Universal Robots PolyScope program: LE02_50.urp

Program LE02_50 (installation=default directory=/programs/LE createdIn=5.7.0.90932 lastSavedIn=5.9.1.1031110 robotSerialNumber=20195501059)
Calibrated DH parameters: a=[0.000146, -0.418764, -0.053981, 0.000058, -0.000023, 0]; d=[0.162545, 37.319448, -206.067439, 168.881546, 0.09955, 0.099464]; alpha=[1.57004, -0.001979, 0.002304, 1.570607, -1.57066, 0]; deltaTheta=[0, -0.174616, -1.258233, 1.432844, -0.000001, 0]
BeforeStart
  'Rev 2021_12_02am 01'
  URCap Gripper Activate (Robotiq_Grippers, Robotiq Inc.) dataModel(ResetAndActivateKey=false)
  start_pose := get_actual_tcp_pose()
  MoveJ speed 60 deg/s, acceleration 80 deg/s^2 (useActiveTCP=true) feature=Base
    Waypoint Waypoint (Variable): variable=start_pose
Robot Program (runOnlyOnce=true)
  'Rev 2021_12_02am 01'
  MoveL speed 250 mm/s, acceleration 1200 mm/s^2 (useActiveTCP=true) feature=Base
    Waypoint Vertical_1: TCP in base x=296.586 y=-399.638 z=157.461 mm, rx=0.0001 ry=0 rz=-0.0068 rad; joints [110.998, -87.379, 110.673, -113.28, 270.04, 201.399] deg; TCP offset x=0 y=0 z=175 mm, rx=3.1416 ry=0 rz=0 rad
    Waypoint Tilted_2: TCP in base x=296.604 y=-399.668 z=157.504 mm, rx=-0.5593 ry=0.007 rz=-0.0068 rad; joints [119.721, -93.557, 131.941, -156.668, 254.371, 206.211] deg
    Set DigitalOutput pin=digital_out[2]; digitalValue=1
    Wait Sleep waitTime=1
    Set DigitalOutput pin=digital_out[2]; digitalValue=0
    Waypoint Vertical_2: TCP in base x=296.586 y=-399.638 z=157.461 mm, rx=0.0001 ry=0 rz=-0.0068 rad; joints [110.998, -87.379, 110.673, -113.28, 270.04, 201.399] deg
    response := "50 success"
